// TIA Portal V20 export
TYPE "UDT_DigSlot"
// DI/DQ module slot
   STRUCT
      Enable : Bool;
      StartAddr : UInt;
      ChannelCount : USInt;
      Reserved : USInt;
   END_STRUCT;
END_TYPE
